PROGRAM GetSpeedSteer
VAR
	steerString : STRING;
	pedalString : STRING;
END_VAR

IF FIND(STR1:= 'Steer', STR2:= RunTCP.sCommand) = 1 THEN
	steerString := RunTCP.sCommand;
ELSIF FIND(STR1:= 'Throttle', STR2:= RunTCP.sCommand) = 1 THEN
	pedalString := RunTCP.sCommand;
END_IF

END_PROGRAM

(* stored: Version 1.1.0.1, ProductVersion 3.1.4024.3
   POU GetSpeedSteer: Id {878004fa-332a-49b4-9634-12c0e2cc0141}, SpecialFunc None *)
